// TIA Portal V16 export
// export: Created 2024-09-05T17:40:14.6329366Z, ExportSetting WithDefaults, DisplayName Totally Integrated Automation Portal, DisplayVersion V16 Update 6, DisplayName TIA Portal Version Control Interface, DisplayVersion V16 Update 2, DisplayName TIA Portal Openness, DisplayVersion V16 Update 6, DisplayName STEP 7 Professional, DisplayVersion V16 Update 6, DisplayName STEP 7 Safety, DisplayVersion V16, DisplayName WinCC Advanced, DisplayVersion V16 Update 6
TYPE "UDT_FittingParameters"
// stored: IsFailsafeCompliant false
   STRUCT
      DigiforceProgram : Int;
      FinalSpeed : Real;
      ApproachSpeed : Real;
      FinalForce : Real;
      ApproachForce : Real;
      EndWayImmediate : Real;   // relative position from digiforce
      EndWayWithTimeout : Real;   // relative position from digiforce
      SwitchingWay : Real;   // absolute cylinder position
      EndWayTimeout : Time;
   END_STRUCT;
END_TYPE
